INTERFACE I_PushButton

PROPERTY IsPressed : BOOL
GET
END_GET
END_PROPERTY

PROPERTY PUBLIC IsReleased : BOOL
GET
END_GET
END_PROPERTY

END_INTERFACE

(* stored: Version 1.1.0.1, ProductVersion 3.1.4024.11
   Itf I_PushButton: Id {f87f46db-800b-4f10-b683-e2b78a381f9d}
   Property IsPressed: Id {d23e84cc-42f4-43d7-a979-be76169e7148}
   Get Get: Id {7803e858-915b-485b-a50b-7ee46db84baf}
   Property IsReleased: Id {c01394d3-16ce-40c4-bd8e-7a47196fbed4}
   Get Get: Id {c27c51aa-d409-4f9e-8eca-bff3a90ddece} *)
